PROGRAM P_Demo_FB_XmlDomParser_InsertChild
VAR
    fbParser : FB_XmlDomParser; // 父 FB 实例
    n : SXmlNode;
    before : SXmlNode;
    name : STRING(255);
    vRet : SXmlNode; // 返回值监视
    bTrigger : BOOL := FALSE; // 在线置 TRUE 触发一次调用
    bTriggerPrev : BOOL;
END_VAR

// =============================================================================
// 场景：在 `FB_XmlDomParser` 的工作流程里完成一个具体子操作；通常配合本 FB 的其他方法组合使用。
// 价值：作为 `FB_XmlDomParser` API 的一部分提供标准化能力，业务代码无需自实现。
// 验证：登录 PLC 在线写 bTrigger := TRUE 触发，monitor 返回值/输出参数。具体步骤见下方注释。
// 验证步骤：
//   1. 右键 PLC 项目下 POUs 文件夹 → Add → Existing Item → 选本 .TcPOU 文件
//   2. 引用 Tc3_JsonXml（References → Add library）
//   3. 编译 → 登录 → 运行；按 verify 注释里给出的在线写值操作
// =============================================================================

// 上升沿触发一次方法调用并观察输出。
IF bTrigger AND NOT bTriggerPrev THEN
    vRet := fbParser.InsertChild(
        n := n,
        before := before,
        name := name
    );
END_IF;
bTriggerPrev := bTrigger;

END_PROGRAM

(* stored: Version 1.1.0.1, ProductVersion 3.1.4024.5
   POU P_Demo_FB_XmlDomParser_InsertChild: Id {109a5486-6ba4-5e58-96f1-9ccec1cbbe0e}, SpecialFunc None *)
